{attribute addProperty BoxType "EJ7342-0000-0019"}
{attribute addProperty Id "VelocityAT %Q*INT162"}
{attribute addProperty CRC "495564226"}
{attribute addProperty SizeInBites "16"}
{attribute addProperty SizeInBytes "2"}
TYPE DCM_Velocity_Channel_1D89B5C2 :
STRUCT
	{attribute addProperty Name "Velocity"}
	Velocity AT %Q* : INT;
END_STRUCT
END_TYPE

(* stored: Version 1.2.0.0, ProductVersion 3.1.4024.9
   DUT DCM_Velocity_Channel_1D89B5C2: Id {a77c4836-770a-4539-9a2f-4d4d1f64c56f} *)
